// TIA Portal V20 export
FUNCTION_BLOCK "LER_SoftCam_Interface_JH"   // FB7, LAD
// stored: Access Published, MemoryReserve 100, SetENOAutomatically false
   VAR_INPUT
      cmsetPositions { ExternalAccessible := 'False'; ExternalVisible := 'False'; ExternalWritable := 'False'} : Array[0..63] of "LBC_typeAxis64PosSetPosition";
      cmMonitoringActualPosition { ExternalAccessible := 'False'; ExternalVisible := 'False'; ExternalWritable := 'False'} : LReal;
      cmConfigTargetposition : LReal;
      cmSelectSetPosition { ExternalAccessible := 'False'; ExternalVisible := 'False'; ExternalWritable := 'False'} : SInt;
      enble : Bool;
      axis : DB_ANY;
   END_VAR
   VAR_OUTPUT
      SoftcamStatus : "emSoftcamInterface";
   END_VAR
   VAR_IN_OUT
      SoftcamListAxisHmi : "LER_typeSoftCamInterface";
   END_VAR
   VAR_TEMP
      LoopCount : Int;
      TempIndex : SInt;
   END_VAR
BEGIN

REGION Network 1: TempIndex
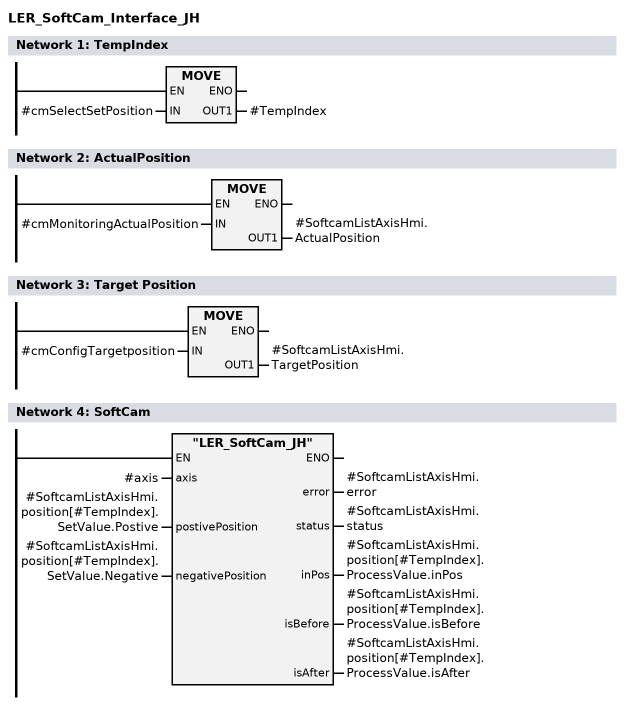
   RUNG wire#powerrail
      Move(in := #cmSelectSetPosition, out1 => #TempIndex)
   END_RUNG
   // the same network as SCL:
   #TempIndex := #cmSelectSetPosition;
END_REGION

REGION Network 2: ActualPosition
   RUNG wire#powerrail
      Move(in := #cmMonitoringActualPosition, out1 => #SoftcamListAxisHmi.ActualPosition)
   END_RUNG
   // the same network as SCL:
   #SoftcamListAxisHmi.ActualPosition := #cmMonitoringActualPosition;
END_REGION

REGION Network 3: Target Position
   RUNG wire#powerrail
      Move(in := #cmConfigTargetposition, out1 => #SoftcamListAxisHmi.TargetPosition)
   END_RUNG
   // the same network as SCL:
   #SoftcamListAxisHmi.TargetPosition := #cmConfigTargetposition;
END_REGION

REGION Network 4: SoftCam
   RUNG wire#powerrail
      "LER_SoftCam_JH"(axis := #axis, postivePosition := #SoftcamListAxisHmi.position[#TempIndex].SetValue.Postive, negativePosition := #SoftcamListAxisHmi.position[#TempIndex].SetValue.Negative, error => #SoftcamListAxisHmi.error, status => #SoftcamListAxisHmi.status, inPos => #SoftcamListAxisHmi.position[#TempIndex].ProcessValue.inPos, isBefore => #SoftcamListAxisHmi.position[#TempIndex].ProcessValue.isBefore, isAfter => #SoftcamListAxisHmi.position[#TempIndex].ProcessValue.isAfter)
   END_RUNG
   // the same network as SCL:
   "LER_SoftCam_JH"(axis := #axis,
                    postivePosition := #SoftcamListAxisHmi.position[#TempIndex].SetValue.Postive,
                    negativePosition := #SoftcamListAxisHmi.position[#TempIndex].SetValue.Negative,
                    error => #SoftcamListAxisHmi.error,
                    status => #SoftcamListAxisHmi.status,
                    inPos => #SoftcamListAxisHmi.position[#TempIndex].ProcessValue.inPos,
                    isBefore => #SoftcamListAxisHmi.position[#TempIndex].ProcessValue.isBefore,
                    isAfter => #SoftcamListAxisHmi.position[#TempIndex].ProcessValue.isAfter);
END_REGION

REGION Network 5 (SCL): FOR Pos
   // sw_cam of Position axis

   #SoftcamListAxisHmi.position[0].ProcessValue.SetPos := #cmsetPositions[0].position;
   #SoftcamListAxisHmi.position[1].ProcessValue.SetPos := #cmsetPositions[1].position;
   #SoftcamListAxisHmi.position[2].ProcessValue.SetPos := #cmsetPositions[2].position;
   #SoftcamListAxisHmi.position[3].ProcessValue.SetPos := #cmsetPositions[3].position;
   #SoftcamListAxisHmi.position[4].ProcessValue.SetPos := #cmsetPositions[4].position;
   #SoftcamListAxisHmi.position[5].ProcessValue.SetPos := #cmsetPositions[5].position;
   #SoftcamListAxisHmi.position[6].ProcessValue.SetPos := #cmsetPositions[6].position;
   #SoftcamListAxisHmi.position[7].ProcessValue.SetPos := #cmsetPositions[7].position;
   #SoftcamListAxisHmi.position[8].ProcessValue.SetPos := #cmsetPositions[8].position;

   // InPos
   FOR #LoopCount := 0 TO 8 DO
       IF #enble AND (#cmMonitoringActualPosition > #SoftcamListAxisHmi.position[#LoopCount].SetValue.Postive) AND (#cmMonitoringActualPosition < #SoftcamListAxisHmi.position[#LoopCount].SetValue.Negative) AND #SoftcamStatus.Softcam.inPos THEN
           #SoftcamStatus.Softcam.InPosSignals[#LoopCount] := true;
       ELSE
           #SoftcamStatus.Softcam.InPosSignals[#LoopCount] := FALSE;
       END_IF;
   END_FOR;
   // PosNo
   FOR #LoopCount := 0 TO 8 DO
       IF #SoftcamStatus.Softcam.InPosSignals[#LoopCount] THEN
           #SoftcamStatus.Softcam.PosNo := INT_TO_DINT((#LoopCount));
       END_IF;
   END_FOR;
END_REGION
END_FUNCTION_BLOCK
